FUNCTION_BLOCK LogWriter (* Extracted Composite Function Block Type *)
  (* Version 11/2/2016, chivdan *)
  PACKAGE Main;
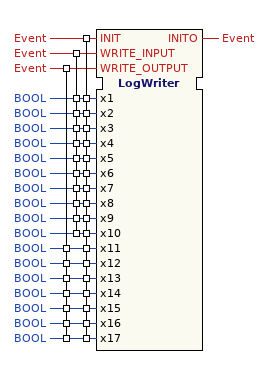
  EVENT_INPUT
    INIT WITH x1, x2, x3, x4, x5, x6, x7, x8, x9, x10, x11, x12, x13, x14, x15, x16, x17; (* Initialization request *)
    WRITE_INPUT WITH x1, x2, x3, x4, x5, x6, x7, x8, x9, x10; (* Normal Execution Request *)
    WRITE_OUTPUT WITH x11, x12, x13, x14, x15, x16, x17;
  END_EVENT
  EVENT_OUTPUT
    INITO;
  END_EVENT
  VAR_INPUT
    x1 : BOOL; (* Argument *)
    x2 : BOOL; (* Argument *)
    x3 : BOOL; (* Argument *)
    x4 : BOOL; (* Argument *)
    x5 : BOOL; (* Argument *)
    x6 : BOOL; (* Argument *)
    x7 : BOOL; (* Argument *)
    x8 : BOOL; (* Argument *)
    x9 : BOOL; (* Argument *)
    x10 : BOOL; (* Argument *)
    x11 : BOOL;
    x12 : BOOL;
    x13 : BOOL;
    x14 : BOOL;
    x15 : BOOL;
    x16 : BOOL;
    x17 : BOOL;
  END_VAR
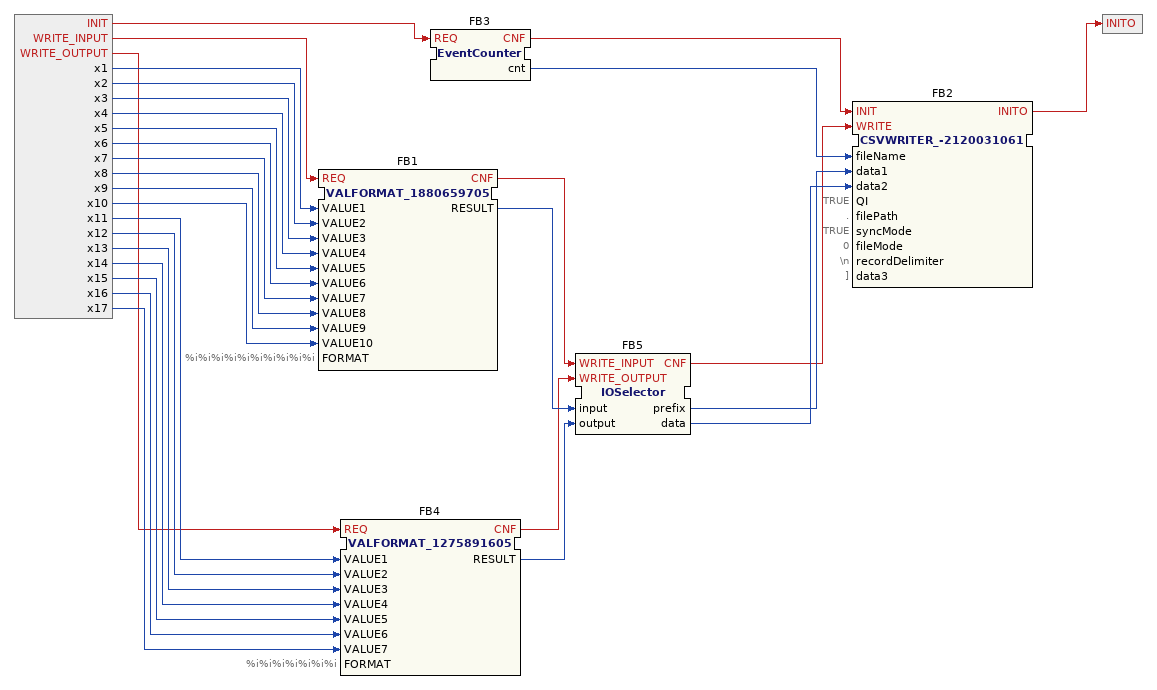
  FBS
    FB2 : CSVWRITER_-2120031061(QI := TRUE, filePath := ., syncMode := TRUE, fileMode := 0, recordDelimiter := \n, data3 := ]); {SET_ATTRIBUTE(Configuration.GenericFBType.InterfaceParams, nxtControl.Standard#I:=3;data${I$}:STRING,STRING,STRING)}
    FB3 : EventCounter;
    FB1 : VALFORMAT_1880659705(FORMAT := %i%i%i%i%i%i%i%i%i%i); {SET_ATTRIBUTE(Configuration.GenericFBType.InterfaceParams, Runtime.Standard#I:=10;VALUE${I$}:INT,INT,INT,INT,INT,INT,INT,INT,INT,INT)}
    FB4 : VALFORMAT_1275891605(FORMAT := %i%i%i%i%i%i%i); {SET_ATTRIBUTE(Configuration.GenericFBType.InterfaceParams, Runtime.Standard#I:=7;VALUE${I$}:INT,INT,INT,INT,INT,INT,INT)}
    FB5 : IOSelector;
  END_FBS
  EVENT_CONNECTIONS
    INIT TO FB3.REQ;
    WRITE_INPUT TO FB1.REQ;
    WRITE_OUTPUT TO FB4.REQ;
    FB1.CNF TO FB5.WRITE_INPUT;
    FB4.CNF TO FB5.WRITE_OUTPUT;
    FB3.CNF TO FB2.INIT;
    FB5.CNF TO FB2.WRITE;
    FB2.INITO TO INITO;
  END_CONNECTIONS
  DATA_CONNECTIONS
    x1 TO FB1.VALUE1;
    x2 TO FB1.VALUE2;
    x3 TO FB1.VALUE3;
    x4 TO FB1.VALUE4;
    x5 TO FB1.VALUE5;
    x6 TO FB1.VALUE6;
    x7 TO FB1.VALUE7;
    x8 TO FB1.VALUE8;
    x9 TO FB1.VALUE9;
    x10 TO FB1.VALUE10;
    x11 TO FB4.VALUE1;
    x12 TO FB4.VALUE2;
    x13 TO FB4.VALUE3;
    x14 TO FB4.VALUE4;
    x15 TO FB4.VALUE5;
    x16 TO FB4.VALUE6;
    x17 TO FB4.VALUE7;
    FB1.RESULT TO FB5.input;
    FB4.RESULT TO FB5.output;
    FB3.cnt TO FB2.fileName;
    FB5.prefix TO FB2.data1;
    FB5.data TO FB2.data2;
  END_CONNECTIONS
END_FUNCTION_BLOCK
